ABB RobotStudio station: Proyecto_Final_B2_20210607-125714.rsstn

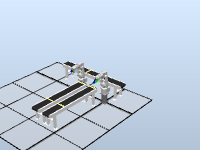
Station Station (saved by RobotStudio 20.4.9280.0)
Layout (positions relative to the parent item):
  - Conveyor_Cuchara [part]
  - Conveyor_Tenedor [part]
  - Conveyor_Caja [part]
  - Caja [part] at (-446, -1910, 506) mm
  - Cuchara [part] at (1969.94, -257.72, 505.09) mm, rotated rx 8.99 ry 0.06 rz 0 deg
  - Tenedor [part] at (1970, -630.69, 506.5) mm
  - Logica_Conveyor_Caja [smart component]
      connections:
        LineSensor_Caja1.SensorOut -> Source_Caja.Execute
        LineSensor_Caja2.SensorOut -> PhysicsControl_Caja.SurfaceVelocityEnabled
    - LineSensor_Caja1 [smart component, from Components\LineSensor.rslib]
        properties: Start=[-0.59 -1 0.515]; End=[-0.31 -1 0.515]; Radius=0.005; SensedPart=(none); SensedPoint=[0 0 0]
      - _sensorPart_ [part]
    - Source_Caja [smart component, from Components\Source.rslib]
        properties: Source=Caja; Copy=(none); Parent=(none); Position=[-0.446 -1.91 0.506]; Orientation=[0 0 0]; Transient=true; PhysicsBehavior=3
    - LineSensor_Caja2 [smart component, from Components\LineSensor.rslib]
        properties: Start=[-0.59 -0.5 0.515]; End=[-0.31 -0.5 0.515]; Radius=0.005; SensedPart=(none); SensedPoint=[0 0 0]
      - _sensorPart_ [part]
    - PhysicsControl_Caja [smart component, from Components\PhysicsControl.rslib]
        properties: Object=Conveyor_Caja; Behavior=1; SurfaceVelocity=0.3
  - Logica_Conveyor_Cuchara [smart component]
      connections:
        LineSensor_Cuchara1.SensorOut -> Source_Cuchara.Execute
        LineSensor_Cuchara2.SensorOut -> PhysicsControl_Cuchara.SurfaceVelocityEnabled
    - LineSensor_Cuchara1 [smart component, from Components\LineSensor.rslib]
        properties: Start=[1.5 -0.39 0.508]; End=[1.5 -0.11 0.508]; Radius=0.003; SensedPart=(none); SensedPoint=[0 0 0]
      - _sensorPart_ [part]
    - Source_Cuchara [smart component, from Components\Source.rslib]
        properties: Source=Cuchara; Copy=(none); Parent=(none); Position=[1.969989 -0.257716 0.505016]; Orientation=[0 0 0]; Transient=true; PhysicsBehavior=3
    - LineSensor_Cuchara2 [smart component, from Components\LineSensor.rslib]
        properties: Start=[0.25 -0.39 0.508]; End=[0.25 -0.11 0.508]; Radius=0; SensedPart=(none); SensedPoint=[0 0 0]
      - _sensorPart_ [part]
    - PhysicsControl_Cuchara [smart component, from Components\PhysicsControl.rslib]
        properties: Object=Conveyor_Cuchara; Behavior=1; SurfaceVelocity=0.3
  - Logica_Conveyor_Tenedor [smart component]
      connections:
        LineSensor_Tenedor.SensorOut -> Source_Tenedor.Execute
        LineSensor_3.SensorOut -> PhysicsControl_Tenedor.SurfaceVelocityEnabled
    - LineSensor_Tenedor [smart component, from Components\LineSensor.rslib]
        properties: Start=[1.5 -0.8 0.508]; End=[1.5 -0.52 0.508]; Radius=0.003; SensedPart=(none); SensedPoint=[0 0 0]
      - _sensorPart_ [part]
    - Source_Tenedor [smart component, from Components\Source.rslib]
        properties: Source=Tenedor; Copy=(none); Parent=(none); Position=[1.97 -0.630694 0.506505]; Orientation=[0 0 0]; Transient=true; PhysicsBehavior=3
    - LineSensor_3 [smart component, from Components\LineSensor.rslib]
        properties: Start=[0.25 -0.8 0.508]; End=[0.25 -0.52 0.508]; Radius=0; SensedPart=(none); SensedPoint=[0 0 0]
      - _sensorPart_ [part]
    - PhysicsControl_Tenedor [smart component, from Components\PhysicsControl.rslib]
        properties: Object=Conveyor_Tenedor; Behavior=1; SurfaceVelocity=0.3
  - IRB120_3_58__01 [mechanism, from Robots\IRB120_3_58_G_01.rslib] at (0, 0, 300) mm; joint values [0, 0, 0, 0, 0.5236, 0] (rad or m)
  - IRB120_3_58__01_2 [mechanism, from Robots\IRB120_3_58_G_01.rslib] at (0, -900, 300) mm; joint values [0, 0, 0, 0, 0.5236, 0] (rad or m)
  - Base_R_Cuchara [part] at (0, -900, 0) mm
  - Base_R_Tenedor [part]
  - Mi_Ventosa [smart component, from Proyecto local\1217c23c-7d3e-48fb-b7d3-d1b2005a3c2bMi_Ventosa.rslib] at (364.35, 0, 894) mm, rotated rx 180 ry 60 rz 180 deg
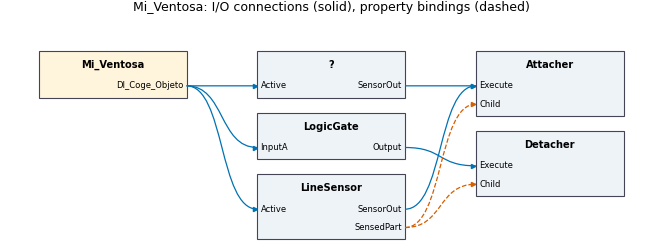
      connections:
        Mi_Ventosa.DI_Coge_Objeto -> ?.Active
        ?.SensorOut -> Attacher.Execute
        Mi_Ventosa.DI_Coge_Objeto -> LogicGate.InputA
        LogicGate.Output -> Detacher.Execute
        Mi_Ventosa.DI_Coge_Objeto -> LineSensor.Active
        LineSensor.SensorOut -> Attacher.Execute
        LineSensor.SensedPart => Attacher.Child
        LineSensor.SensedPart => Detacher.Child
    - Attacher [smart component, from Components\Attacher.rslib]
        properties: Parent=Ventosa; Flange=0; Child=(none); Mount=false; Offset=[0 0 0]; Orientation=[0 0 0]
    - Detacher [smart component, from Components\Detacher.rslib]
        properties: Child=(none); KeepPosition=true
    - Ventosa [mechanism, from Proyecto local\1217c23c-7d3e-48fb-b7d3-d1b2005a3c2bMi_Ventosa.rslib] at (0, 0, 0) mm
    - LogicGate [smart component, from Components\LogicGate.rslib]
        properties: Operator=NOT; Delay=0
    - LineSensor [smart component, from Components\LineSensor.rslib]
        properties: Start=[0 0 0.055]; End=[0 0 0.07]; Radius=0.001; SensedPart=(none); SensedPoint=[0 0 0]
      - _sensorPart_ [part, from Proyecto local\1217c23c-7d3e-48fb-b7d3-d1b2005a3c2bMi_Ventosa.rslib]
    - Indicador [part, from Proyecto local\1217c23c-7d3e-48fb-b7d3-d1b2005a3c2bMi_Ventosa.rslib] at (-4.38, 0, 0) mm
Attachment: Mi_Ventosa is attached to IRB120_3_58__01 / Link6
Targets, tools, work objects and paths stored in the station, written as RAPID:
! task (no controller)
MODULE CalibData
  PERS tooldata TCP_Ventosa:=[TRUE,[[0,0,60],[1,0,0,0]],[0.1,[0,0,1],[1,0,0,0],0,0,0]];
ENDMODULE

